// Monitors the dump chiller from the flow sensor
FUNCTION_BLOCK FB_DumpChiller
VAR_INPUT
	bAmphosOn : BOOL; // Whether the amphos is turned on
	bDumpChillerFlow : BOOL; // Signal from the flow sensor. Normally high.
	bMasterLatchReset : BOOL; //Master latched error reset
END_VAR
VAR_OUTPUT
	{attribute 'pytmc' := '
		pv: ERROR
		io: i
		field: OSV MAJOR
		field: ZSV NO_ALARM
		field: ZNAM OK
		field: ONAM ERROR
	'}
	bError : BOOL; // Whether an error was detected. Latches until reset
END_VAR
VAR
END_VAR

(* Latch error if the dump chiller flow detects an error and the amphos is on *)
IF bAmphosOn AND NOT bDumpChillerFlow THEN
	bError := TRUE;
END_IF

IF bMasterLatchReset THEN
	bError := FALSE;
END_IF

// Reset latched errors
METHOD Reset
VAR_INPUT
END_VAR
bError := FALSE;
END_METHOD

END_FUNCTION_BLOCK

(* stored: Version 1.1.0.1, ProductVersion 3.1.4024.6
   POU FB_DumpChiller: Id {e80bbd01-109d-4f0c-b0c9-7110d73e1445}, SpecialFunc None
   Method Reset: Id {9ead59f4-c71a-4d56-be28-6cfd674dd28b} *)
